PROGRAM MAIN
VAR
    sDevSTate : STRING;
    iSampleToRun : UINT := 0;
END_VAR

sDevSTate := F_ScannerDevStateToString(IO.ScannerDevState);

CASE iSampleToRun OF
    0:
        PRG_SimpleExample();
    1:
        PRG_ExtendedExample();
	2:
		PRG_KepwareExample();
END_CASE

END_PROGRAM

(* stored: Version 1.1.0.1, ProductVersion 3.1.4024.12
   POU MAIN: Id {3cede1a2-b51a-40dc-8ef9-feea4f37dd90}, SpecialFunc None *)
